Universal Robots PolyScope program: halt_83.urp

Program halt_83 (createdIn=3.2.19293 lastSavedIn=3.2.19293 directory=/programs installation=default robotSerialNumber=2015351391)
Calibrated DH parameters: a=[0.000352, -0.161198, -0.373486, 0.00005, 0.000049, 0]; d=[0.089268, 352.477598, -320.08558, -32.281492, 0.094939, 0.082518]; alpha=[1.570728, 0.001116, -0.003686, 1.571189, -1.570572, 0]; deltaTheta=[-0.000012, 1.181849, -1.491165, 0.309495, -0.000007, 0.000025]
Robot Program (runOnlyOnce=false motionType=MoveJ speed=1.047198 acceleration=1.396263 recalculateMotions=false)
  MoveL speed 250 mm/s, acceleration 1200 mm/s^2 (recalculateMotions=false) feature=Base
    Waypoint waypoint1: TCP in base x=160.931 y=198.845 z=524.744 mm, rx=-1.5849 ry=-0.1114 rz=-0.2806 rad; joints [73.055, -56.065, -125.506, 0.863, 100.732, -14.67] deg
    Waypoint waypoint2 (Relative): motionParameters(blendRadius=0); relativeFromPosition TCP in base x=160.927 y=198.835 z=524.759 mm, rx=-1.5849 ry=-0.1114 rz=-0.2806 rad; joints [73.055, -56.068, -125.508, 0.862, 100.735, -14.671] deg; TCP in base x=460.008 y=198.847 z=524.759 mm, rx=-1.5849 ry=-0.1114 rz=-0.2806 rad; joints [28.367, -98.878, -92.612, 10.027, 145.495, -15.624] deg
    Waypoint waypoint3 (Relative): relativeFromPosition TCP in base x=460.014 y=198.837 z=524.74 mm, rx=-1.585 ry=-0.1114 rz=-0.2806 rad; joints [28.367, -98.878, -92.612, 10.027, 145.495, -15.624] deg; TCP in base x=460.025 y=198.822 z=323.999 mm, rx=-1.585 ry=-0.1113 rz=-0.2805 rad; joints [28.334, -111.086, -109.601, 39.335, 145.618, -15.483] deg
    Waypoint waypoint4 (Relative): relativeFromPosition TCP in base x=460.016 y=198.817 z=324.002 mm, rx=-1.585 ry=-0.1113 rz=-0.2805 rad; joints [28.334, -111.086, -109.601, 39.335, 145.618, -15.483] deg; TCP in base x=159.997 y=198.837 z=323.981 mm, rx=-1.585 ry=-0.1114 rz=-0.2804 rad; joints [73.267, -70.988, -150.726, 41.013, 100.654, -14.57] deg
    Halt
